Yaskawa INFORM job: -90_90.JBI

/JOB
//NAME -90_90
///FOLDERNAME OBROTNIK
//POS
///NPOS 0,0,1,0,0,0
///TOOL 0
///POSTYPE PULSE
///PULSE
EC00000=-798154,556474
//INST
///DATE 2023/11/07 19:00
///ATTR SC,RW,RJ
////FRAME ROBOT
///GROUP1 ST1
NOP
MOVJ EC00000 VJ=100.00
END
